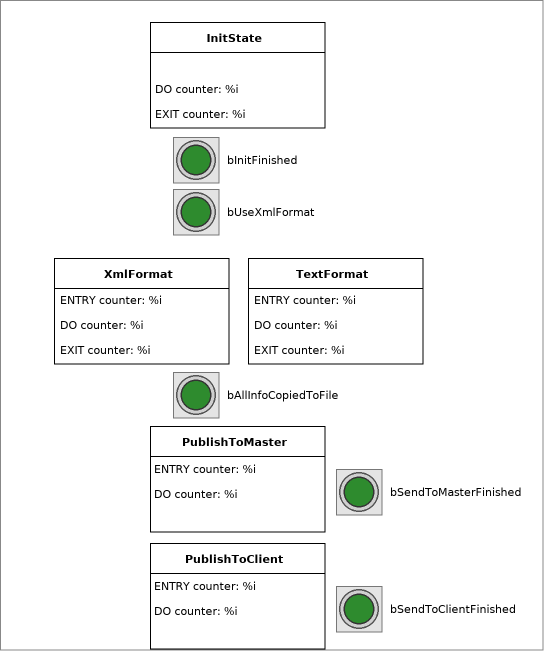
VISUALIZATION Visu_Composite  // 544x651
    Rectangle (150,22 175x106)
    Line (150,52) (325,52)
    Label (152,27 165x23), "InitState"
    Rectangle (54,258 175x106)
    Line (54,288) (229,288)
    Label (56,263 165x23), "XmlFormat"
    Rectangle (248,258 175x106)
    Line (248,288) (423,288)
    Label (250,263 165x23), "TextFormat"
    Rectangle (150,426 175x106)
    Line (150,456) (325,456)
    Label (152,431 165x23), "PublishToMaster"
    Rectangle (150,543 175x106)
    Line (150,573) (325,573)
    Label (152,548 165x23), "PublishToClient"
    PushSwitch (173,137 46x46), variable: MAIN.fbUmlSc.bInitFinished, behaviour: TOGGLE, style: Switch-PushSwitch-Green
    Label (224,149 118x23), "bInitFinished"
    PushSwitch (173,189 46x46), variable: MAIN.fbUmlSc.bUseXmlFormat, behaviour: TOGGLE, style: Switch-PushSwitch-Green
    Label (224,201 118x23), "bUseXmlFormat"
    PushSwitch (173,372 46x46), variable: MAIN.fbUmlSc.bAllInfoCopiedToFile, behaviour: TOGGLE, style: Switch-PushSwitch-Green
    Label (224,384 137x23), "bAllInfoCopiedToFile"
    PushSwitch (336,469 46x46), variable: MAIN.fbUmlSc.bSendToMasterFinished, behaviour: TOGGLE, style: Switch-PushSwitch-Green
    Label (387,481 155x23), "bSendToMasterFinished"
    PushSwitch (336,586 46x46), variable: MAIN.fbUmlSc.bSendToClientFinished, behaviour: TOGGLE, style: Switch-PushSwitch-Green
    Label (387,598 141x23), "bSendToClientFinished"
    Rectangle (152,54 169x21), text variable: GVL.nCounterInit
    Rectangle (152,79 169x21), "DO counter: %i", text variable: GVL.nCounterInit
    Rectangle (152,104 169x21), "EXIT counter: %i", text variable: GVL.nCounterSaveInitSettings
    Rectangle (57,290 169x21), "ENTRY counter: %i", text variable: GVL.nCounterClearXml
    Rectangle (57,315 169x21), "DO counter: %i", text variable: GVL.nCounterFillXml
    Rectangle (57,340 169x21), "EXIT counter: %i", text variable: GVL.nCounterSaveXml
    Rectangle (251,290 169x21), "ENTRY counter: %i", text variable: GVL.nCounterClearText
    Rectangle (251,315 169x21), "DO counter: %i", text variable: GVL.nCounterFillText
    Rectangle (251,340 169x21), "EXIT counter: %i", text variable: GVL.nCounterSaveText
    Rectangle (151,459 169x21), "ENTRY counter: %i", text variable: GVL.nCounterGetMasterID
    Rectangle (151,484 169x21), "DO counter: %i", text variable: GVL.nCounterSendToMaster
    Rectangle (151,509 169x21), text variable: GVL.nCounterInit
    Rectangle (151,576 169x21), "ENTRY counter: %i", text variable: GVL.nCounterGetClientID
    Rectangle (151,601 169x21), "DO counter: %i", text variable: GVL.nCounterSendToClient
    Rectangle (151,626 169x21), text variable: GVL.nCounterInit
END_VISUALIZATION

(* stored: Version 1.1.0.1
   Visu Visu_Composite: Id {3956f65f-b89c-4520-b21f-37dff8c3becc} *)
